Omron CX-Programmer project NewProject (CX-Programmer 9.61)

# PLC NewPLC1: CJ2H CPU65-EIP
I/O table (CPU CJ2H-CPU65-EIP): rack 0 slot 11 CJ2B-EIP21

## Global symbols (name address type ; comment)
10.00 BOOL  ; RELAY1
0.00 BOOL  ; TOMBOL ON
0.01 BOOL  ; TOMBOL OFF
10.01 BOOL  ; LAMPU 1

## Program NewProgram1 (cyclic task 0)

### Section Section1

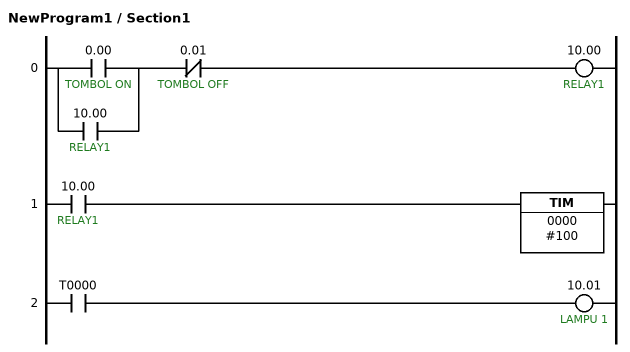
; rung 0
LD 0.00  ; TOMBOL ON
OR 10.00  ; RELAY1
ANDNOT 0.01  ; TOMBOL OFF
OUT 10.00  ; RELAY1
; rung 1
LD 10.00  ; RELAY1
TIM 0000 #100
; rung 2
LD T0000
OUT 10.01  ; LAMPU 1

### Section END
; rung 0
END(001)